(* CODESYS project codesys

Project tree, tasks and I/O mapping:
  Device : EC44, Epec Oy, order no. n/a, version 3.5.13.66
    application Application
      task MainTask (cyclic, interval t#10ms, priority 1) calls PLC_PRG
      program PLC_PRG [ST]
    io_interface : io_interface, Epec, order no. n/a, version 3.5.13.66
        unmapped channels: , , , , , , , , , , , , , , , , , , , , , , , , , , , , , , , , , , , , , , , ,
          , , , , , , , , , , , , , , , , , , , , , , , , , , , , , , , , , , , , , , , ,
          , , , , , , , , , , , , , , , , , , , , , , , , , , , , , , , , , , , , , , , ,
          , , , , , , , , , , , , , , , , , , , , , , , , , , , , , , , , , , , , , , , ,
          , , , , , , , , , , , , , , , , , , , , , , , , , , , , , , , , , , , , , , , ,
          , , , , , , , , 
*)

// Device/Application/PLC_PRG
PROGRAM PLC_PRG
VAR
	a:INT;
	b:INT;
	c:INT;
	
END_VAR

a:= 1;
b:=2;
C:= a+b;

END_PROGRAM
